// TIA Portal project "CommRS485" (V17)

(* hardware
DEVICE "Station S7-1200_2"  S7-1200 Station
   slot 0: "Châssis_0"  S7-1200 Rack  Rack  V1.0
   slot 1: "PLC_Esclave"  CPU 1215C AC/DC/Rly  6ES7 215-1BG31-0XB0  V3.0
   slot 101: "CM 1241 (RS485)_1"  CM 1241 (RS485)  6ES7 241-1CH30-0XB0  V1.0
DEVICE "Station S7-1200_1"  S7-1200 Station
   slot 0: "Châssis_0"  S7-1200 Rack  Rack  V1.0
   slot 1: "PLC_Maitre"  CPU 1211C DC/DC/Rly  6ES7 211-1HE40-0XB0  V4.5
   slot 101: "CM 1241 (RS422/485)_1"  6ES7 241-1CH32-0XB0  V2.2
*)

// ===== PLC "PLC_Maitre"  CPU 1211C DC/DC/Rly =====

VAR_GLOBAL   // PLC tag table "Table de variables standard"
   "System_Byte" AT %MB0 : Byte;
   "FirstScan" AT %M0.0 : Bool;
   "DiagStatusUpdate" AT %M0.1 : Bool;
   "AlwaysTRUE" AT %M0.2 : Bool;
   "AlwaysFALSE" AT %M0.3 : Bool;
   "Clock_Byte" AT %MB1 : Byte;
   "Clock_10Hz" AT %M1.0 : Bool;
   "Clock_5Hz" AT %M1.1 : Bool;
   "Clock_2.5Hz" AT %M1.2 : Bool;
   "Clock_2Hz" AT %M1.3 : Bool;
   "Clock_1.25Hz" AT %M1.4 : Bool;
   "Clock_1Hz" AT %M1.5 : Bool;
   "Clock_0.625Hz" AT %M1.6 : Bool;
   "Clock_0.5Hz" AT %M1.7 : Bool;
   "MODE_MASTER" AT %M2.0 : Bool;
   "scanOne" AT %M2.1 : Bool;
   "Tag_1" AT %M4.0 : Bool;
   "Mode_SLAVE" AT %M4.1 : Bool;
END_VAR

DATA_BLOCK "MBLOAD"   // DB1
{ S7_Optimized_Access := 'FALSE' }
VERSION : 0.1
   VAR
      Baud : UDInt := 9600;
      PARITY : UInt;
      DONE : Bool;
      ERROR : Bool;
      STATUS : Word;
   END_VAR
BEGIN
END_DATA_BLOCK

DATA_BLOCK "MBCONFIG"   // DB2
{ S7_Optimized_Access := 'FALSE' }
VERSION : 0.1
   VAR
      REQ : Bool;
      AGAIN : Bool;
      MB_ADDR : UInt := 1;   // DEFAULT ADRESS : 1
      MODE : USInt;   // READ ONLY : 0
      DATA_ADDR : UDInt := 10001;   // STARTING ADRESS : 40001
      DATA_LEN : UInt := 10;   // DATA LENGTH : 10 WORDS
      DONE : Bool;
      ERROR : Bool;
      BUSY : Bool;
      Register_Input : Array[0..9] of Bool;
      STATUS : Word;
   END_VAR
BEGIN
END_DATA_BLOCK

DATA_BLOCK "DATA_BUFF"   // DB3
{ S7_Optimized_Access := 'FALSE' }
VERSION : 0.1
   VAR
      REGISTERS : Array[0..9] of Bool;
   END_VAR
BEGIN
END_DATA_BLOCK

FUNCTION "REQ_Master_To_Slave" : Void   // FC1, LAD
{ S7_Optimized_Access := 'TRUE' }
VERSION : 0.1
BEGIN

REGION Network 1
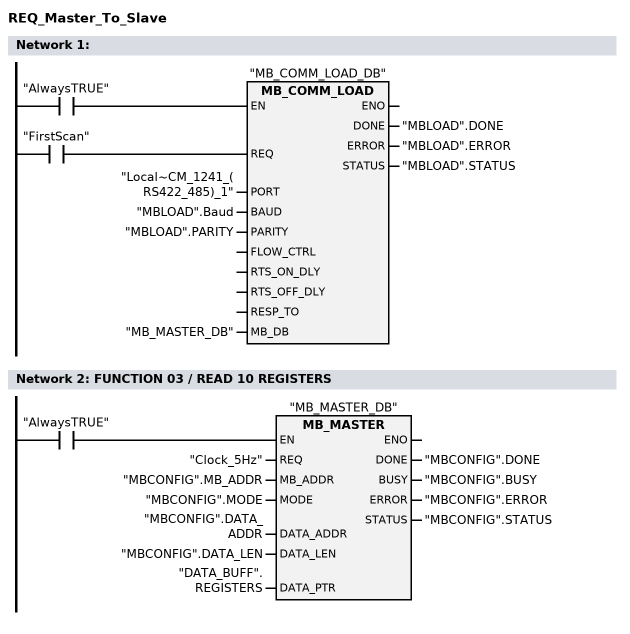
   IF "AlwaysTRUE" THEN
       "MB_COMM_LOAD_DB"(REQ := "FirstScan",   // MB_COMM_LOAD
                         PORT := "Local~CM_1241_(RS422_485)_1",
                         BAUD := "MBLOAD".Baud,
                         PARITY := "MBLOAD".PARITY,
                         MB_DB := "MB_MASTER_DB",
                         DONE => "MBLOAD".DONE,
                         ERROR => "MBLOAD".ERROR,
                         STATUS => "MBLOAD".STATUS);
   END_IF;
END_REGION

REGION Network 2: FUNCTION 03 / READ 10 REGISTERS
   IF "AlwaysTRUE" THEN
       "MB_MASTER_DB"(REQ := "Clock_5Hz",   // MB_MASTER
                      MB_ADDR := "MBCONFIG".MB_ADDR,
                      MODE := "MBCONFIG".MODE,
                      DATA_ADDR := "MBCONFIG".DATA_ADDR,
                      DATA_LEN := "MBCONFIG".DATA_LEN,
                      DATA_PTR := "DATA_BUFF".REGISTERS,
                      DONE => "MBCONFIG".DONE,
                      BUSY => "MBCONFIG".BUSY,
                      ERROR => "MBCONFIG".ERROR,
                      STATUS => "MBCONFIG".STATUS);
   END_IF;
END_REGION
END_FUNCTION

FUNCTION "REQ_Slave_To_Master" : Void   // FC2, LAD
{ S7_Optimized_Access := 'TRUE' }
VERSION : 0.1
   VAR_TEMP   // added for the SCL form of the ladder/FBD networks
      _w1 : Bool;
   END_VAR
BEGIN

REGION Network 1
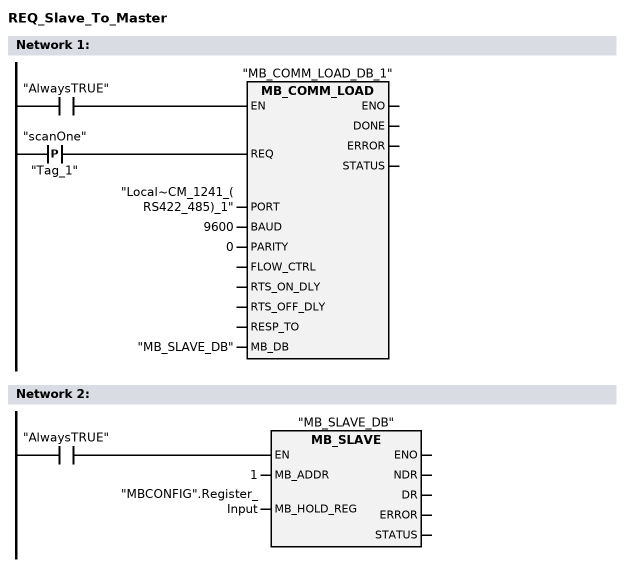
   #_w1 := "scanOne" AND NOT "Tag_1";   // rising edge of "scanOne"
   "Tag_1" := "scanOne";
   IF "AlwaysTRUE" THEN
       "MB_COMM_LOAD_DB_1"(REQ := #_w1,   // MB_COMM_LOAD
                           PORT := "Local~CM_1241_(RS422_485)_1",
                           BAUD := 9600,
                           PARITY := 0,
                           MB_DB := "MB_SLAVE_DB");
   END_IF;
END_REGION

REGION Network 2
   IF "AlwaysTRUE" THEN
       "MB_SLAVE_DB"(MB_ADDR := 1, MB_HOLD_REG := "MBCONFIG".Register_Input);   // MB_SLAVE
   END_IF;
END_REGION
END_FUNCTION

ORGANIZATION_BLOCK "Main"   // OB1, LAD, ProgramCycle
TITLE = "Main Program Sweep (Cycle)"
{ S7_Optimized_Access := 'TRUE' }
VERSION : 0.1
   VAR_INPUT
      Initial_Call : Bool;   // Initial call of this OB
      Remanence : Bool;   // =True, if remanent data are available
   END_VAR
BEGIN

REGION Network 1: Call Request Master To Slave
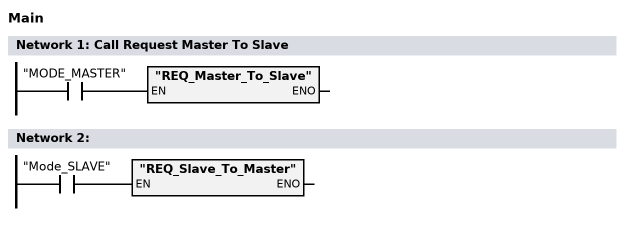
   RUNG wire#powerrail
      Contact( "MODE_MASTER" )
      "REQ_Master_To_Slave"()
   END_RUNG
   // the same network as SCL:
   IF "MODE_MASTER" THEN "REQ_Master_To_Slave"(); END_IF;
END_REGION

REGION Network 2
   RUNG wire#powerrail
      Contact( "Mode_SLAVE" )
      "REQ_Slave_To_Master"()
   END_RUNG
   // the same network as SCL:
   IF "Mode_SLAVE" THEN "REQ_Slave_To_Master"(); END_IF;
END_REGION
END_ORGANIZATION_BLOCK

// ===== PLC "PLC_Esclave"  CPU 1215C AC/DC/Rly =====

VAR_GLOBAL   // PLC tag table "Table de variables standard"
   "System_Byte" AT %MB1 : Byte;
   "FirstScan" AT %M1.0 : Bool;
   "DiagStatusUpdate" AT %M1.1 : Bool;
   "AlwaysTRUE" AT %M1.2 : Bool;
   "AlwaysFALSE" AT %M1.3 : Bool;
   "Clock_Byte" AT %MB0 : Byte;
   "Clock_10Hz" AT %M0.0 : Bool;
   "Clock_5Hz" AT %M0.1 : Bool;
   "Clock_2.5Hz" AT %M0.2 : Bool;
   "Clock_2Hz" AT %M0.3 : Bool;
   "Clock_1.25Hz" AT %M0.4 : Bool;
   "Clock_1Hz" AT %M0.5 : Bool;
   "Clock_0.625Hz" AT %M0.6 : Bool;
   "Clock_0.5Hz" AT %M0.7 : Bool;
END_VAR

DATA_BLOCK "MBLOAD"   // DB1
{ S7_Optimized_Access := 'FALSE' }
VERSION : 0.1
   VAR
      BAUD : UDInt := 9600;
      PARITY : UInt;
      DONE : Bool;
      ERROR : Bool;
      STATUS : Word;
   END_VAR
BEGIN
END_DATA_BLOCK

DATA_BLOCK "MBCONFIG"   // DB2
{ S7_Optimized_Access := 'FALSE' }
VERSION : 0.1
   VAR
      MB_ADDR : UInt := 1;
      ERROR : Bool;
      Static_7 : Bool;
      STATUS : Word;
      NDR : Bool;
      DR : Bool;
   END_VAR
BEGIN
END_DATA_BLOCK

DATA_BLOCK "DATA_BUFF"   // DB3
{ S7_Optimized_Access := 'FALSE' }
VERSION : 0.1
   VAR
      REGISTERS : Array[0..9] of Int;
   END_VAR
BEGIN
END_DATA_BLOCK

ORGANIZATION_BLOCK "Main"   // OB1, LAD, ProgramCycle
TITLE = "Main Program Sweep (Cycle)"
{ S7_Optimized_Access := 'TRUE' }
VERSION : 0.1
BEGIN

REGION Network 1
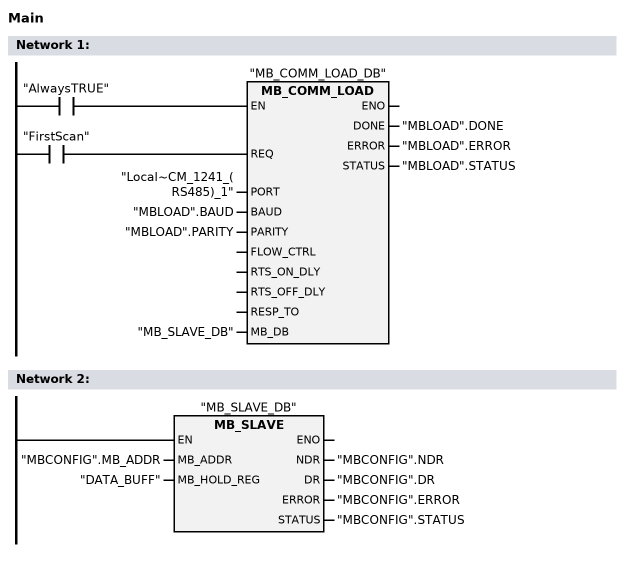
   IF "AlwaysTRUE" THEN
       "MB_COMM_LOAD_DB"(REQ := "FirstScan",   // MB_COMM_LOAD
                         PORT := "Local~CM_1241_(RS485)_1",
                         BAUD := "MBLOAD".BAUD,
                         PARITY := "MBLOAD".PARITY,
                         MB_DB := "MB_SLAVE_DB",
                         DONE => "MBLOAD".DONE,
                         ERROR => "MBLOAD".ERROR,
                         STATUS => "MBLOAD".STATUS);
   END_IF;
END_REGION

REGION Network 2
   "MB_SLAVE_DB"(MB_ADDR := "MBCONFIG".MB_ADDR,   // MB_SLAVE
                 MB_HOLD_REG := "DATA_BUFF",
                 NDR => "MBCONFIG".NDR,
                 DR => "MBCONFIG".DR,
                 ERROR => "MBCONFIG".ERROR,
                 STATUS => "MBCONFIG".STATUS);
END_REGION
END_ORGANIZATION_BLOCK